(* IEC 61131-3 sources: RL_MAR/experiments/comparison/autoplc/results/deepseek-ai-DeepSeek-V3.2_20260508_111905/hf_20, 1 file *)

(* ---- hf_20_1.st ---- *)
FUNCTION_BLOCK FB_ProductionLineControl
VAR_INPUT
    Mode : BOOL; // Manual/Auto mode selection
    ForwardButton : BOOL; // Forward rotation button
    ReverseButton : BOOL; // Reverse rotation button
    SensorA : BOOL; // Sensor A input
    SensorB : BOOL; // Sensor B input
    SensorC : BOOL; // Sensor C input
    ButtonA : BOOL; // Button A input
    ButtonB : BOOL; // Button B input
    ButtonC : BOOL; // Button C input
END_VAR

VAR_OUTPUT
    MotorForward : BOOL; // Motor forward output
    MotorReverse : BOOL; // Motor reverse output
    CompletionLight : BOOL; // Process completion indicator
END_VAR

VAR
    State : INT; // State machine current state
END_VAR

// Main execution logic
IF State = 0 THEN
    // Initialization state
    MotorForward := FALSE;
    MotorReverse := FALSE;
    CompletionLight := FALSE;
    State := 1;
END_IF;

IF NOT Mode THEN
    // Manual Mode Operation
    // Forward motion condition
    IF ForwardButton AND NOT ReverseButton THEN
        MotorForward := TRUE;
        MotorReverse := FALSE;
    // Reverse motion condition
    ELSIF ReverseButton AND NOT ForwardButton THEN
        MotorForward := FALSE;
        MotorReverse := TRUE;
    // Stop condition (both buttons pressed or neither pressed)
    ELSE
        MotorForward := FALSE;
        MotorReverse := FALSE;
    END_IF;

    // CompletionLight remains off in manual mode
    CompletionLight := FALSE;
ELSE
    // Automatic Mode Operation
    CASE State OF
        1: // State 1: Waiting at Station A
            MotorForward := FALSE;
            MotorReverse := FALSE;
            IF SensorA THEN
                State := 2;
            END_IF;

        2: // State 2: Processing at Station A
            MotorForward := FALSE;
            MotorReverse := FALSE;
            IF ButtonA THEN
                MotorForward := TRUE;
                MotorReverse := FALSE;
                State := 3;
            END_IF;

        3: // State 3: Moving to Station B
            // MotorForward remains TRUE from previous state
            MotorReverse := FALSE;
            IF SensorB THEN
                MotorForward := FALSE;
                State := 4;
            END_IF;

        4: // State 4: Processing at Station B
            MotorForward := FALSE;
            MotorReverse := FALSE;
            IF ButtonB THEN
                MotorForward := TRUE;
                MotorReverse := FALSE;
                State := 5;
            END_IF;

        5: // State 5: Moving to Station C
            // MotorForward remains TRUE from previous state
            MotorReverse := FALSE;
            IF SensorC THEN
                MotorForward := FALSE;
                State := 6;
            END_IF;

        6: // State 6: Processing at Station C
            MotorForward := FALSE;
            MotorReverse := FALSE;
            IF ButtonC THEN
                CompletionLight := TRUE;
                State := 7;
            END_IF;

        7: // State 7: Cycle Completion
            MotorForward := FALSE;
            MotorReverse := FALSE;
            IF NOT SensorC THEN
                CompletionLight := FALSE;
                State := 1;
            END_IF;
    END_CASE;
END_IF;

END_FUNCTION_BLOCK
